TYPE MNG_POSE6 :(* position and orientation as an euler based pose *)
STRUCT
	x, y, z, a, b, c : REAL;
END_STRUCT
END_TYPE

(* stored: Version 1.1.0.1, ProductVersion 3.1.0.23
   DUT MNG_POSE6: Id {a8469f91-805b-4695-af22-93a030cc974b} *)
